{attribute 'qualified_only'}
{attribute 'strict'}
TYPE PtWeekDay :
(
	MONDAY := 0,
    TUESDAY := 1,
    WEDNESDAY := 2,
    THURSDAY := 3,
    FRIDAY := 4,
    SATURDAY := 5,
    SUNDAY := 6
);
END_TYPE

(* stored: Version 1.1.0.1, ProductVersion 3.1.4024.12
   EnumerationTextList PtWeekDay: Id {d13310af-7732-460b-aa4e-5247a3499f0c} *)
